{attribute 'linkalways'} 
{attribute 'no_explicit_call' := 'This FB is a CLASS and must be accessed using methods or properties'}
{attribute 'enable_dynamic_creation'}
FUNCTION_BLOCK Node_F_VN_GenerateAffineTransformationUnitMatrix2D EXTENDS VisionNode
VAR
    aTransformationMatrix : _TcVnMatrix2x3_LREAL;
    hrPrev : _HRESULT(S_OK);
	hresult : _HRESULT(S_OK);
END_VAR

METHOD PUBLIC  Clone : I_Node
VAR
	pNode : POINTER TO Node_F_VN_GenerateAffineTransformationUnitMatrix2D;
END_VAR
pNode := __NEW(Node_F_VN_GenerateAffineTransformationUnitMatrix2D);
Clone := pNode^;
END_METHOD

METHOD FB_init : BOOL
VAR_INPUT
	bInitRetains : BOOL; // if TRUE, the retain variables are initialized (warm start / cold start)
	bInCopyCode : BOOL;  // if TRUE, the instance afterwards gets moved into the copy code (online change)
END_VAR
AddInput('hrPrev', hrPrev);
AddOutput('aTransformationMatrix', aTransformationMatrix);
AddOutput('hresult',hresult);
END_METHOD

METHOD PROTECTED OnExecute
hresult.Value := F_VN_GenerateAffineTransformationUnitMatrix2D(
	aTransformationMatrix := aTransformationMatrix.Value,
	hrPrev := hrPrev.Value);
END_METHOD

METHOD PUBLIC PreExecutionCheck
VAR_INPUT
	Check : I_PreExecutionChecks;
END_VAR
END_METHOD

END_FUNCTION_BLOCK

(* stored: Version 1.1.0.1, ProductVersion 3.1.4024.13
   POU Node_F_VN_GenerateAffineTransformationUnitMatrix2D: Id {16183bcf-9e78-0442-3508-2455d3458b19}, SpecialFunc None
   Folder Constructor: Id {84bd84f2-3fc4-07fa-220d-1a4658d16f98}
   Method Clone: Id {a4315591-3b39-0dd6-39db-d9a1ff414291}
   Method FB_init: Id {69b5de50-7068-090e-2922-4be58d6f2a31}
   Method OnExecute: Id {a24b83fc-1fd0-0973-1123-551204ac53fe}
   Method PreExecutionCheck: Id {de843bb3-1f03-0df4-276c-0766050316ff} *)
